// TIA Portal V17 export
// export: Created 2023-12-22T15:04:42.1924801Z, ExportSetting WithDefaults, DisplayName Totally Integrated Automation Portal, DisplayVersion V17, DisplayName TIA Portal Openness, DisplayVersion V17, DisplayName TIA Portal Version Control Interface, DisplayVersion V17, DisplayName STEP 7 Professional, DisplayVersion V17, DisplayName STEP 7 Safety, DisplayVersion V17, DisplayName WinCC Advanced, DisplayVersion V17
DATA_BLOCK "DIx_1_DB"   // DB200
VERSION : 0.1
// stored: AutoNumber false, DBAccessibleFromOPCUA true, InstanceOfName DIx_1, InstanceOfType FB
"DIx_1"
   // VAR RETAIN
   //    AllBlock { S7_SetPoint := 'True'} : "DI_ex";
   //    "3FOk" { S7_SetPoint := 'True'} : "DI_ex";
   //    Pump_Alarm { S7_SetPoint := 'True'} : "DI_ex";
   //    Leak_KP { S7_SetPoint := 'True'} : "DI_ex";
   //    Level_Norm { S7_SetPoint := 'True'} : "DI_ex";
   //    "3Fok_1" { S7_SetPoint := 'True'} : "DI_ex";
   //    "3Fok_2" { S7_SetPoint := 'True'} : "DI_ex";
   //    "3Fok_sh" { S7_SetPoint := 'True'} : "DI_ex";
   //    SHUSKV_Ok { S7_SetPoint := 'True'} : "DI_ex";
   //    Leak_KP_res { S7_SetPoint := 'True'} : "DI_ex";
   //    Leak_KP_res_1 { S7_SetPoint := 'True'} : "DI_ex";
   //    signal_12 { S7_SetPoint := 'True'} : "DI_ex";
   //    Time_DTL { S7_SetPoint := 'True'} : DTL := DTL#2012-01-22-23:24:13.460664;
   // END_VAR
BEGIN
   AllBlock.Use.Inverse := FALSE;
   AllBlock.Use.Indirect := TRUE;
   AllBlock.ADDR_Byte := 0;
   AllBlock.ADDR_Bit := 3;
   AllBlock.Filter_On.SP := 16#02;
   AllBlock.Filter_Off.SP := 16#02;
   "3FOk".Use.Inverse := FALSE;
   "3FOk".Use.Indirect := TRUE;
   "3FOk".ADDR_Byte := 0;
   "3FOk".ADDR_Bit := 0;
   "3FOk".Filter_On.SP := 16#02;
   "3FOk".Filter_Off.SP := 16#02;
   Pump_Alarm.Use.Inverse := FALSE;
   Pump_Alarm.Use.Indirect := TRUE;
   Pump_Alarm.ADDR_Byte := 0;
   Pump_Alarm.ADDR_Bit := 2;
   Pump_Alarm.Filter_On.SP := 16#02;
   Pump_Alarm.Filter_Off.SP := 16#02;
   Leak_KP.Use.Inverse := FALSE;
   Leak_KP.Use.Indirect := TRUE;
   Leak_KP.ADDR_Byte := 0;
   Leak_KP.ADDR_Bit := 4;
   Leak_KP.Filter_On.SP := 16#02;
   Leak_KP.Filter_Off.SP := 16#02;
   Level_Norm.Use.Inverse := FALSE;
   Level_Norm.Use.Indirect := TRUE;
   Level_Norm.ADDR_Byte := 0;
   Level_Norm.ADDR_Bit := 5;
   Level_Norm.Filter_On.SP := 16#02;
   Level_Norm.Filter_Off.SP := 16#02;
   "3Fok_1".Use.Inverse := FALSE;
   "3Fok_1".Use.Indirect := TRUE;
   "3Fok_1".ADDR_Byte := 0;
   "3Fok_1".ADDR_Bit := 6;
   "3Fok_1".Filter_On.SP := 16#02;
   "3Fok_1".Filter_Off.SP := 16#02;
   "3Fok_2".Use.Inverse := FALSE;
   "3Fok_2".Use.Indirect := TRUE;
   "3Fok_2".ADDR_Byte := 0;
   "3Fok_2".ADDR_Bit := 7;
   "3Fok_2".Filter_On.SP := 16#02;
   "3Fok_2".Filter_Off.SP := 16#02;
   "3Fok_sh".Use.Inverse := FALSE;
   "3Fok_sh".Use.Indirect := TRUE;
   "3Fok_sh".ADDR_Byte := 1;
   "3Fok_sh".ADDR_Bit := 0;
   "3Fok_sh".Filter_On.SP := 16#02;
   "3Fok_sh".Filter_Off.SP := 16#02;
   SHUSKV_Ok.Use.Inverse := FALSE;
   SHUSKV_Ok.Use.Indirect := TRUE;
   SHUSKV_Ok.ADDR_Byte := 1;
   SHUSKV_Ok.ADDR_Bit := 1;
   SHUSKV_Ok.Filter_On.SP := 16#02;
   SHUSKV_Ok.Filter_Off.SP := 16#02;
   Leak_KP_res.Use.Inverse := FALSE;
   Leak_KP_res.Use.Indirect := TRUE;
   Leak_KP_res.ADDR_Byte := 1;
   Leak_KP_res.ADDR_Bit := 2;
   Leak_KP_res.Filter_On.SP := 16#02;
   Leak_KP_res.Filter_Off.SP := 16#02;
   Leak_KP_res_1.Use.Inverse := FALSE;
   Leak_KP_res_1.Use.Indirect := TRUE;
   Leak_KP_res_1.ADDR_Byte := 1;
   Leak_KP_res_1.ADDR_Bit := 3;
   Leak_KP_res_1.Filter_On.SP := 16#02;
   Leak_KP_res_1.Filter_Off.SP := 16#02;
   signal_12.Use.Inverse := FALSE;
   signal_12.Use.Indirect := TRUE;
   signal_12.ADDR_Byte := 0;
   signal_12.ADDR_Bit := 9;
   signal_12.Filter_On.SP := 16#02;
   signal_12.Filter_Off.SP := 16#02;
END_DATA_BLOCK
